FUNCTION Convert_DT_TO_ULINT : Hresult
VAR_INPUT
	in : DT;
	out : REFERENCE TO ULINT;
END_VAR
VAR
	converted : ULINT;
END_VAR

converted := DT_TO_ULINT(in);

IF (ULINT_TO_DT(converted) <> in) THEN
	Convert_DT_TO_ULINT := INCOMPATIBLE;
	RETURN;
END_IF

out := converted;

END_FUNCTION

(* stored: Version 1.1.0.1, ProductVersion 3.1.4024.12
   POU Convert_DT_TO_ULINT: Id {0b3fe122-ea99-43cd-b156-85a7921d7122}, SpecialFunc None *)
